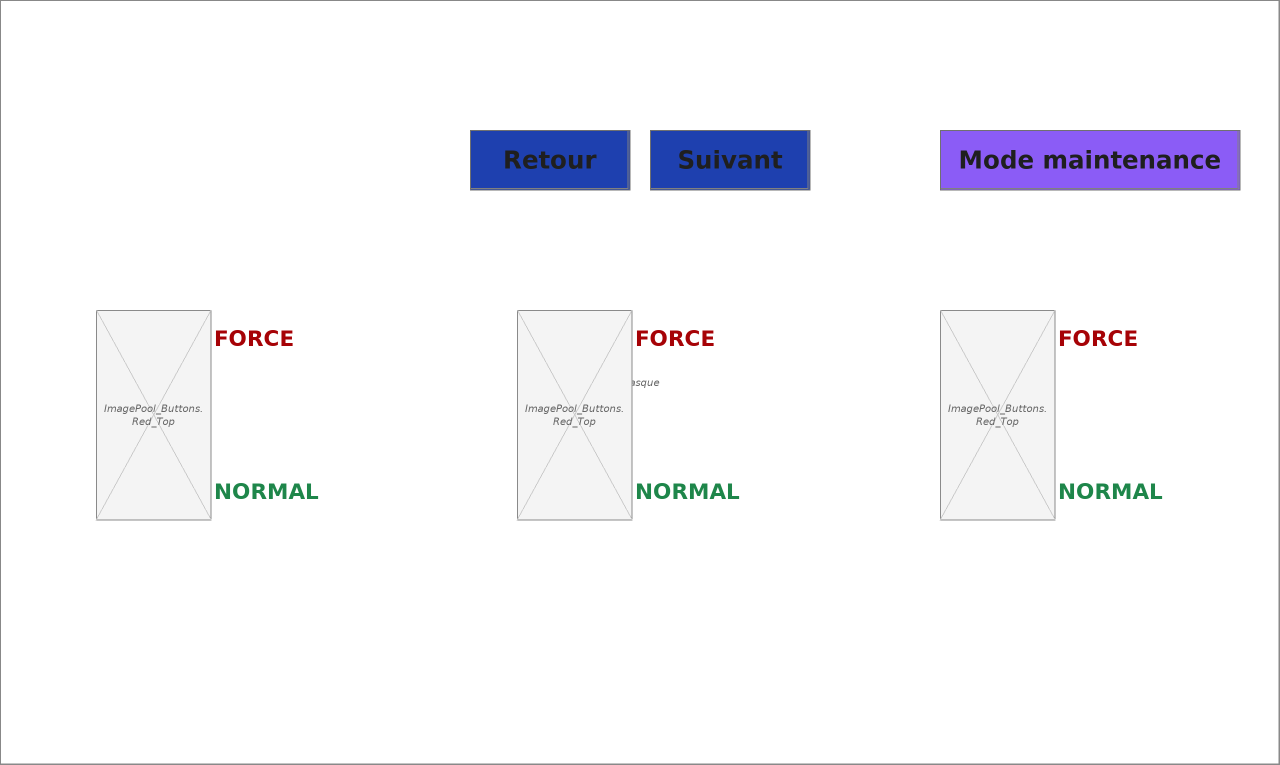
VISUALIZATION Maintenance_1  // 1280x765
    Frame (0,0 1280x765)
        shows masque()
    Button (470,130 160x60), "Retour"
        OnMouseDown: change screen: menu
        OnMouseDown: VisuUserMgmt Type=Logout
    Button (940,130 300x60), "Mode maintenance"
        OnMouseDown: toggle Cmd_Mode_Maintenance
    Group (445,246 390x500), invisible if: NOT Option_RegSouf_Ultrason
        Rectangle (3,0 380x76), "Soufflage"
        RoundedRectangle (0,272 390x76), "Débit : %d m3/h", text variable: F_Cons_Registre_Soufflage, invisible if: NOT EF_Cons_Registre_Soufflage
            OnMouseDown: write the text variable via VisuDialogs.Numpad, min 0, max 1000, format %d
        Rectangle (0,349 390x76), "Appli : %.0f m3/h", text variable: Cons_Actio_Registre_Souf_m3h
        Rectangle (0,424 390x76), "Mesure : %.0f m3/h", text variable: Tab_MES_Sonde_Gros_Debit_Soufflage.R_MesCor
        Group (72,64 246x208)
            Group (0,0 115x210)
                Image (0,0 115x210), invisible if: EF_Cons_Registre_Soufflage, image: ImagePool_Buttons.Green_Bottom
                    OnMouseDown: toggle EF_Cons_Registre_Soufflage
                Image (0,0 115x210), invisible if: NOT EF_Cons_Registre_Soufflage, image: ImagePool_Buttons.Red_Top
                    OnMouseDown: toggle EF_Cons_Registre_Soufflage
            Rectangle (115,0 132x57), "FORCE"
            Rectangle (112,76 132x57), "MODE"
            Rectangle (115,153 132x57), "NORMAL"
    Button (650,130 160x60), "Suivant"
        OnMouseDown: execute {
            IF (Option_Douche OR Option_Lavabo)
            	THEN
            	VisuElems.CURRENTVISU := 'Maintenance_2';
            	ELSIF (Option_Bas_Debit OR Option_Douchette OR Option_NEP)
            		THEN
            		VisuElems.CURRENTVISU := 'Maintenance_3';
            	ELSIF (Option_WC_GV OR Option_WC_PV OR Option_Prise)
            		THEN
            		VisuElems.CURRENTVISU := 'Maintenance_4';
            	ELSIF (Option_Cabine_Climatique)
            		THEN
            		VisuElems.CURRENTVISU := 'Maintenance_5';
            	ELSIF (Option_Com_RegSouf_Ultrason)
            		THEN
            		VisuElems.CURRENTVISU := 'Maintenance_6';
            	ELSE
            		VisuElems.CURRENTVISU := 'Maintenance_7';
            END_IF
        }
    Group (24,246 390x500)
        Rectangle (3,0 380x76), "Extraction"
        Group (72,64 246x208)
            Group (0,0 115x210)
                Image (0,0 115x210), invisible if: EF_Cons_Reg_Etanche_Ext, image: ImagePool_Buttons.Green_Bottom
                    OnMouseDown: toggle EF_Cons_Reg_Etanche_Ext
                Image (0,0 115x210), invisible if: NOT EF_Cons_Reg_Etanche_Ext, image: ImagePool_Buttons.Red_Top
                    OnMouseDown: toggle EF_Cons_Reg_Etanche_Ext
            Rectangle (115,0 132x57), "FORCE"
            Rectangle (112,76 132x57), "MODE"
            Rectangle (115,153 132x57), "NORMAL"
        Rectangle (0,349 390x76), "Appli : %.0f %%", text variable: Cons_Actionneur_Reg_Etanche_Ext
        Rectangle (0,424 390x76), "Mesure : %.0f %%", text variable: MES_Pos_Reg_Etanche_Ext
        RoundedRectangle (0,272 390x76), "Ouverture : %.0f %%", text variable: F_Cons_Reg_Etanche_Ext, invisible if: NOT EF_Cons_Reg_Etanche_Ext
            OnMouseDown: write the text variable via VisuDialogs.Numpad, min 0, max 100, format %.0f
    Group (868,246 390x500), invisible if: NOT Option_V3V_EauMitig
        Rectangle (3,0 380x76), "Vanne eau mitigée"
        Group (72,64 246x208)
            Group (0,0 115x210)
                Image (0,0 115x210), invisible if: EF_Cons_V3V_Eau_Mitig, image: ImagePool_Buttons.Green_Bottom
                    OnMouseDown: toggle EF_Cons_V3V_Eau_Mitig
                Image (0,0 115x210), invisible if: NOT EF_Cons_V3V_Eau_Mitig, image: ImagePool_Buttons.Red_Top
                    OnMouseDown: toggle EF_Cons_V3V_Eau_Mitig
            Rectangle (115,0 132x57), "FORCE"
            Rectangle (112,76 132x57), "MODE"
            Rectangle (115,153 132x57), "NORMAL"
        Rectangle (0,349 390x76), "Appli : %.0f %%", text variable: Cons_Actionneur_V3V_Eau_Mitig
        Rectangle (0,424 390x76), "Mesure : %.0f %%", text variable: Cons_Actionneur_V3V_Eau_Mitig, invisible if: TRUE
        RoundedRectangle (0,272 390x76), "Ouverture : %.0f %%", text variable: F_Cons_V3V_Eau_Mitig, invisible if: NOT EF_Cons_V3V_Eau_Mitig
            OnMouseDown: write the text variable via VisuDialogs.Numpad, min 0, max 100, format %.0f
END_VISUALIZATION

(* stored: Version 1.1.0.1, ProductVersion 3.1.4024.15
   Visu Maintenance_1: Id {a08f9dca-9958-48ca-abeb-9a96763f97bc} *)
